PROGRAM TEST
VAR
	TEST_STATE1:TEST_STATE;
	j: INT;
END_VAR

CASE TEST_STATE1 OF
	TEST_0:
		j:=10;
		TEST_STATE1:=TEST_1;
	TEST_1:
		j:=j+10;
END_CASE

END_PROGRAM

(* stored: Version 1.1.0.1, ProductVersion 3.1.4024.0
   POU TEST: Id {43bf10ca-c042-4a96-86d0-577d363b2543}, SpecialFunc None *)
